{attribute 'linkalways'} 
{attribute 'no_explicit_call' := 'This FB is a CLASS and must be accessed using methods or properties'}
{attribute 'enable_dynamic_creation'}
FUNCTION_BLOCK Node_F_VN_AddToContainerElements_SINT EXTENDS VisionNode
VAR
    nValue : _SINT(0);
    ipContainer : _ITcVnContainer;
    hrPrev : _HRESULT(S_OK);
    hresult : _HRESULT(S_OK);
END_VAR

METHOD PUBLIC  Clone : I_Node
VAR
    pNode : POINTER TO Node_F_VN_AddToContainerElements_SINT;
END_VAR
pNode := __NEW(Node_F_VN_AddToContainerElements_SINT);
Clone := pNode^;
END_METHOD

METHOD FB_init : BOOL
VAR_INPUT
    bInitRetains : BOOL; // if TRUE, the retain variables are initialized (warm start / cold start)
    bInCopyCode : BOOL;  // if TRUE, the instance afterwards gets moved into the copy code (online change)
END_VAR
AddParameter('nValue', nValue);
AddInput('ipContainer', ipContainer);
AddInput('hrPrev', hrPrev);
AddOutput('ipContainer', ipContainer);
AddOutput('hresult',hresult);
END_METHOD

METHOD PROTECTED OnExecute
hresult.Value := F_VN_AddToContainerElements_SINT(
    nValue := nValue.Value,
    ipContainer := ipContainer.Value,
    hrPrev:= hrPrev.Value);
END_METHOD

METHOD PUBLIC PreExecutionCheck
VAR_INPUT
    Check : I_PreExecutionChecks;
END_VAR
Check.IsTrue(ipContainer.IsValid, 'ipContainer must be a valid container');
Check.IsTrue(ipContainer.IsType(TC_GLOBAL_CONST_LIST.ContainerType_Vector_SINT), 'ipContainer contains incorrect type');
END_METHOD

END_FUNCTION_BLOCK

(* stored: Version 1.1.0.1, ProductVersion 3.1.4026.13
   POU Node_F_VN_AddToContainerElements_SINT: Id {d6c73595-336d-40d5-880d-4bf3bacb0ae6}, SpecialFunc None
   Folder Constructor: Id {0fc43161-695c-4f41-ae72-18374273c393}
   Method Clone: Id {7c1fbc60-14cf-45ae-a55d-737c834fc7cb}
   Method FB_init: Id {b83deeb1-18a3-4b6a-9cbe-a0b0a6a8aed7}
   Method OnExecute: Id {5bc2a4de-bd1d-4c3e-af58-eb1f53ed80b4}
   Method PreExecutionCheck: Id {2907f614-6cf7-47c1-a4b5-ecfe39ac7d17} *)
